// TIA Portal V20 export
TYPE "type_emRelations_em3"
// stored: Access Published, Namespace Unit1
   STRUCT
      "Bool" { ExternalWritable := 'False'} : Array[0..99] of Bool;
      LReal { ExternalWritable := 'False'} : Array[0..19] of LReal;
      isLinked : Bool;
      softCam : "Unit1.type_emRelations_em3_SoftCam";
      cmStatus { S7_SetPoint := 'True'} : "Unit1.type_emRelations_em3_cmStatus";
      sequence { S7_SetPoint := 'True'} : "Unit1.type_emRelations_em3_sequence";
   END_STRUCT;
END_TYPE
